(* CoDeSys 2.3 export: E_ENUM.EXP *)

(* Data type *)
TYPE E_Enum :
(
	Disabled 	:= 0,
	Starting 		:= 50,
	Running 		:= 100,
	Stopping		:= 200,
	Unknown		:= -99
);
END_TYPE
